# EPICS alarm handler configuration: mps_database/bareTest/alarms/areas/mpln_sps_mp01.alhConfig
GROUP NULL MPLN:SPS:MP01:1
$ALIAS MPS Link Node 191
$GUIDANCE
LTUH MPS
   Group Name: MPLN:SPS:MP01:1
   Summary PV:  MPLN:SPS:MP01:1:STATSUMY
$END
CHANNEL  MPLN:SPS:MP01:1    MPLN:SPS:MP01:1:MPS_EN_RBV		-----
CHANNEL  MPLN:SPS:MP01:1    MPLN:SPS:MP01:1:LC1_MODE_RBV		-----
